# B&R Automation Studio project prac 3
Automation Studio 4.5.2.102

## Configuration Config1

### IoMap.iom - 4PP065_0571_P74/IoMap.iom
```iecst
VAR_CONFIG
	Cyclic#1.gAxis02_DrvIf.iLifeCnt AT %IB."8I64xxxxxxx.00x-1".SDC_LifeCnt;
	Cyclic#1.gAxis02_DrvIf.iDrvOK AT %IX."8I64xxxxxxx.00x-1".ETAD_Input_Bool_02;
	Cyclic#1.gAxis02_DrvIf.oSetTime AT %QW."8I64xxxxxxx.00x-1".SDC_SetTime;
	::Program:speed AT %QW."8I64xxxxxxx.00x-1".LFRD_Output;
	Cyclic#1.gAxis02_DiDoIf.iLifeCntDriveReady AT %IB."8I64xxxxxxx.00x-1".SDC_LifeCnt;
	Cyclic#1.gAxis02_DiDoIf.iLifeCntDriveEnable AT %IB."8I64xxxxxxx.00x-1".SDC_LifeCnt;
	Cyclic#1.gAxis02_DiDoIf.oDriveEnable AT %QX."8I64xxxxxxx.00x-1".CMDD_Output_Bool_00;
	Cyclic#1.gAxis02_ModuleOk AT %QX."8I64xxxxxxx.00x-1".CMDD_Output_Bool_01;
	Cyclic#1.gAxis02_ModuleOk AT %QX."8I64xxxxxxx.00x-1".CMDD_Output_Bool_02;
	Cyclic#1.gAxis02_ModuleOk AT %IX."8I64xxxxxxx.00x-1".ModuleOk;
	Cyclic#1.gAxis02_DiDoIf.oDriveEnable AT %QX."8I64xxxxxxx.00x-1".CMDD_Output_Bool_03;
	Cyclic#1.gAxis02_DiDoIf.iDriveReady AT %IX."8I64xxxxxxx.00x-1".ETAD_Input_Bool_02;
	EVIRD.STATE AT %IW."8I64xxxxxxx.00x-1".ETAD_Input;
	::EVIRD.COM AT %QW."8I64xxxxxxx.00x-1".CMDD_Output;
END_VAR
```

## Logical view

Binary libraries used (declarations not repeated): Library

### Global.var - Global variables
```iecst
VAR
	gAxis01 : ACP10AXIS_typ;
	gAxis01_HW : SdcHwCfg_typ := (0);
	gAxis01_DrvIf : SdcDrvIf16_typ := (0);
	gAxis01_DiDoIf : SdcDiDoIf_typ := (0);
	gAxis01_ModuleOk : BOOL := 0;
	gAxis02 : ACP10AXIS_typ;
	gAxis02_HW : SdcHwCfg_typ := (0);
	gAxis02_DrvIf : SdcDrvIf16_typ := (0);
	gAxis02_DiDoIf : SdcDiDoIf_typ := (0);
	gAxis02_ModuleOk : BOOL := 0;
	EVIRD : DRIVE;
END_VAR
```

Listed in the project but not available here: Logical/Global.typ, Logical/Libraries, Logical/acp10etxen, Logical/Program, Logical/ncsdcctrl, Logical/gAxis01obj, Logical/gAxis02obj
